// Mitsubishi GX Works2 project: 240510_실린더A+-실린더B+-   PLC: Q02U

PROGRAM MAIN
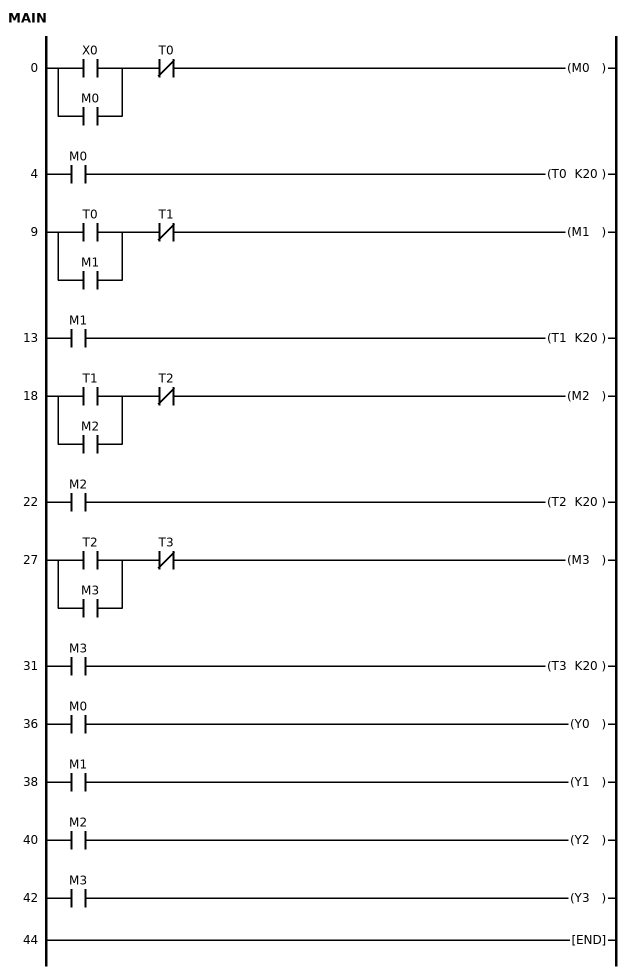
0     LD      X0
      OR      M0
      ANI     T0
      OUT     M0
4     LD      M0
      OUT     T0 K20
9     LD      T0
      OR      M1
      ANI     T1
      OUT     M1
13    LD      M1
      OUT     T1 K20
18    LD      T1
      OR      M2
      ANI     T2
      OUT     M2
22    LD      M2
      OUT     T2 K20
27    LD      T2
      OR      M3
      ANI     T3
      OUT     M3
31    LD      M3
      OUT     T3 K20
36    LD      M0
      OUT     Y0
38    LD      M1
      OUT     Y1
40    LD      M2
      OUT     Y2
42    LD      M3
      OUT     Y3
44    END
END_PROGRAM
